Yaskawa INFORM job: ROVI_SOLVE.JBI

/JOB
//NAME ROVI_SOLVE
///FOLDERNAME ROVI
//POS
///NPOS 0,0,0,0,0,0
//ARGINFO
///ARGTYPE B,,,,,,,
///COMMENT
POS_SHIFT_REG







//INST
///DATE 2020/01/07 16:04
///ATTR SC,RW
///GROUP1 RB1
///LVARS 1,2,0,0,0,0,0,0
NOP
GETARG LB000 IARG#(1)
CALL JOB:CLEAR_POS ARGFLB000
SET LI000 I092
SET LI001 0
*SOLVE
SET I080 90
SET B080 2
WAIT B080=255
INC LI001
IFTHENEXP I080<>0
	 RET I080 IF LI001>=LI000
	 TIMER T=0.500
	 JUMP *SOLVE IF LI000<>0
ENDIF
RET I080
END
